/// Enumeration of possible axis motion commands.
TYPE E_MotionCommand :
(
	/// No command
	eMotionCommand_none := 0,
	/// Reset axis
	eMotionCommand_reset := 1,
	/// Axis halt (default stopping method)
	eMotionCommand_halt := 2,
	/// Axis stop (needs reset before next motion command)
	eMotionCommand_stop := 3,
	/// Axis homing
	eMotionCommand_home := 4,
	/// Set axis position
	eMotionCommand_setPos := 5,
	/// Jog axis
	eMotionCommand_jog := 6,
	/// Jog axis accelerating
	eMotionCommand_jogAcc := 7,
	/// Move axis to point
	eMotionCommand_moveAbs := 8,
	/// Move axis additive
	eMotionCommand_moveAdd := 9,
	/// Move axis relative
	eMotionCommand_moveRel := 10,
	/// Move axis modulo
	eMotionCommand_moveMod := 11,
	/// Move axis velocity (endles)
	eMotionCommand_moveVel := 12,
	/// Apply axis torque
	eMotionCommand_torque := 13,
	/// Gear axis in (electronic) or change gear ratio
	eMotionCommand_gearIn := 14,
	/// Gear axis out (electronic), default behavior: halt axis after gear out
	eMotionCommand_gearOut := 15,
	/// Axis start/stop touch probe
	eMotionCommand_touchProbe := 16,
	/// Force MC reset axis
	eMotionCommand_resetMc := 17,
	/// Group add
	eMotionCommand_GroupAdd := 18,
	/// torque control
	eMotionCommand_torqCtrl := 19,
	
	/// set ax axis position offset
	eMotionCommand_setAxPosOffs := 20
);
END_TYPE

(* stored: Version 1.1.0.1, ProductVersion 3.1.4024.12
   DUT E_MotionCommand: Id {33de73fb-3737-4471-9582-307eef3db450} *)
